// TwinCAT 3 PLC project Libraries
// Title: Logging/file library
// Company: Ziga
// Author: Ziga
// ProjectVersion: 0.0.1.1
// Description: A library containing file/logging functionalities.
// ProgramVersion: 3.1.4024.0
// libraries:
//   Tc2_Standard, * (Beckhoff Automation GmbH)
//   Tc2_System, * (Beckhoff Automation GmbH)
//   Tc2_Utilities, * (Beckhoff Automation GmbH)
//   Tc3_Module, * (Beckhoff Automation GmbH)
//   TcUnit, * (www.tcunit.org)
//   Core, * (Ziga)
// project tree:
//   SOURCE/FileHandler/POUs/ FB_FileHandler.TcPOU, I_FileHandler.TcIO (not stored)
//   SOURCE/Logger/DUTs/ E_LoggerState.TcDUT (not stored)
//   SOURCE/Logger/POUs/ FB_Logger.TcPOU
//   / TestsTask.TcTTO (not stored)
//   TESTS/ PRG_TESTS.TcPOU (not stored)
//   TESTS/Test suites/ FB_FileHandler_Tests.TcPOU (not stored), FB_Logger_Tests.TcPOU
//   Version/ Global_Version.TcGVL (not stored)
// real-time tasks:
//   TASK TestsTask: cycle T#10ms, priority 20, ADS port 350

// ---- SOURCE/FileHandler/POUs/FB_FileHandler.TcPOU
// A function block containing multiple file handling methods.
// For examples refer to tests in the folder "TESTS/Test suites", file "FB_FileHandlerTests".
FUNCTION_BLOCK FB_FileHandler EXTENDS ZigasLibs_Core.FB_ErrorSource IMPLEMENTS I_FileHandler

VAR
	_fileHandle		: UINT;
	_fileProperties	: ZigasLibs_Core.ST_FileProperties;
	_error			: BOOL;
	_amsAddress		: Tc2_System.ST_AmsAddr;
END_VAR

{attribute 'monitoring':='variable'}
(* Gets or sets the Ams address structure*)
PROPERTY AmsAddress : REFERENCE TO ZigasLibs_Core.Tc2_System.ST_AmsAddr
GET
AmsAddress ref= _amsAddress;
END_GET
SET
_amsAddress := AmsAddress;
END_SET
END_PROPERTY

(* Closes the file (if opened). Returns TRUE when done - method needs to be called until it returns TRUE!*)
METHOD PRIVATE Close : BOOL

VAR_INST
	fbFileClose			: Tc2_System.FB_FileClose;
	nCloseFileState		: UINT;
END_VAR

VAR CONSTANT
	FILE_CLOSE_START 		: UINT := 0;
	FILE_CLOSE_WAIT_BUSY	: UINT := 10;
	FILE_CLOSE_DONE			: UINT := 20;
END_VAR
IF THIS^.HandleCreated = FALSE THEN
	Close := TRUE;
	RETURN;
END_IF

_error := _error OR fbFileClose.bError;

CASE nCloseFileState OF
	FILE_CLOSE_START:
		fbFileClose(bExecute := FALSE);
		fbFileClose(bExecute := TRUE, hFile := _fileHandle);
		nCloseFileState := FILE_CLOSE_WAIT_BUSY;
		
	FILE_CLOSE_WAIT_BUSY:
		fbFileClose(bExecute := FALSE);
		IF NOT fbFileClose.bBusy AND NOT fbFileClose.bError THEN
			nCloseFileState := FILE_CLOSE_DONE;
		END_IF

	FILE_CLOSE_DONE:
		Close := TRUE;
		_fileHandle := 0;
		nCloseFileState := FILE_CLOSE_START;
END_CASE

_error := _error OR fbFileClose.bError;
IF fbFileClose.bError THEN
	_errorSource.ErrorCode := fbFileClose.nErrId;
END_IF
END_METHOD

(* Creates the file. Returns TRUE when done - method needs to be called until it returns TRUE!*)
METHOD Create : BOOL
VAR_INPUT
	(* If file already exists, it will be deleted and crated once again (content will be lost!)*)
	bOverwrite	: BOOL;
END_VAR

VAR_INST
	nFileCreateState	: UINT;
END_VAR

VAR CONSTANT
	FILE_CREATE_STATE_START					: UINT := 0;
	FILE_CREATE_STATE_OVERWRITE_OR_CREATE	: UINT := 10;
	FILE_CREATE_STATE_WAIT_DONE				: UINT := 20;
	FILE_CREATE_STATE_DONE					: UINT := 30;
END_VAR
CASE nFileCreateState OF
	FILE_CREATE_STATE_START:
		nFileCreateState := FILE_CREATE_STATE_OVERWRITE_OR_CREATE;
		
	FILE_CREATE_STATE_OVERWRITE_OR_CREATE:
		IF bOverwrite THEN
			IF THIS^.Open(mode := ZigasLibs_Core.E_FileOpenMode.BINARY_READ_WRITE_OVERWRITE_EXISTING) THEN
				nFileCreateState := FILE_CREATE_STATE_WAIT_DONE;
			END_IF
		ELSE
			IF THIS^.Open(mode := ZigasLibs_Core.E_FileOpenMode.BINARY_APPEND) THEN
				nFileCreateState := FILE_CREATE_STATE_WAIT_DONE;
			END_IF
		END_IF
		
	FILE_CREATE_STATE_WAIT_DONE:
		IF THIS^.Close() THEN
			nFileCreateState := FILE_CREATE_STATE_DONE;
		END_IF

	FILE_CREATE_STATE_DONE:
		nFileCreateState := FILE_CREATE_STATE_START;
END_CASE
END_METHOD

(* Deletes the file, if it exists. Returns TRUE when done - method needs to be called until it returns TRUE!*)
METHOD Delete : BOOL

VAR_INST
	fbFileDelete		: Tc2_System.FB_FileDelete;
	FtrigDeleteFinished	: Tc2_Standard.F_TRIG;
	bCheckIfFileExists	: BOOL;
	bFileExists			: BOOL;
END_VAR
fbFileDelete(
	bExecute := NOT fbFileDelete.bBusy,
	sPathName := ZigasLibs_Core.FileHelper.CreateFilePath(_fileProperties.FileLocation, _fileProperties.FileName,  ''));
	
FtrigDeleteFinished(CLK := fbFileDelete.bBusy);
IF FtrigDeleteFinished.Q THEN
	fbFileDelete(bExecute := FALSE);
	Delete := TRUE;
END_IF

_error := _error OR fbFileDelete.bError;
END_METHOD

{attribute 'monitoring':='variable'}
(* Gets the error state, if any of the functions failed.*)
PROPERTY Error : BOOL
GET
Error := _error;
END_GET
END_PROPERTY

(* Checks if the file exists. Returns TRUE when done - method needs to be called until it returns TRUE!*)
METHOD Exists : BOOL
VAR_INPUT
	(* When mehod is finished, the variable provided here will have the result, TRUE if file exists, FALSE if not.*)
	refFileExists	: REFERENCE TO BOOL;
END_VAR

VAR_INST
	fbFileExists			: Tc2_Utilities.FB_EnumFindFileEntry := (tTimeout := T#5S);
	nCheckFileExistState	: UINT;
END_VAR

VAR CONSTANT
	FILE_EXIST_STATE_PREPARE	: UINT := 0;
	FILE_EXIST_STATE_START		: UINT := 10;
	FILE_EXIST_STATE_CHECK		: UINT := 20;
	FILE_EXIST_STATE_DONE		: UINT := 30;
	FILE_EXIST_STATE_ERROR		: uint := 9999;
END_VAR
CASE nCheckFileExistState OF
	FILE_EXIST_STATE_PREPARE:
		fbFileExists(bExecute := FALSE, eCmd := Tc2_Utilities.E_EnumCmdType.eEnumCmd_First);
		refFileExists := FALSE;
		nCheckFileExistState := FILE_EXIST_STATE_START;
		
	FILE_EXIST_STATE_START:
		fbFileExists(bExecute := TRUE,
			sPathName := ZigasLibs_Core.FileHelper.CreateFilePath(_fileProperties.FileLocation, _fileProperties.FileName, ''),
			sNetId := ZigasLibs_Core.AmsHelper.NetIdToString(_amsAddress.netId));
		nCheckFileExistState := FILE_EXIST_STATE_CHECK;
	
	FILE_EXIST_STATE_CHECK:
		fbFileExists(bExecute := FALSE);
		IF NOT fbFileExists.bBusy THEN
			IF NOT fbFileExists.bError THEN
				IF fbFileExists.stFindFile.sFileName = _fileProperties.FileName THEN
					refFileExists := TRUE;
					nCheckFileExistState := FILE_EXIST_STATE_DONE;
				END_IF	
				IF NOT fbFileExists.bEOE THEN
					fbFileExists.eCmd := Tc2_Utilities.E_EnumCmdType.eEnumCmd_Next;
				ELSE
					refFileExists := FALSE;
					nCheckFileExistState := FILE_EXIST_STATE_DONE;
				END_IF
			ELSE
				nCheckFileExistState := FILE_EXIST_STATE_ERROR;
			END_IF
		END_IF
	
	FILE_EXIST_STATE_DONE:
		Exists := TRUE;
		nCheckFileExistState := FILE_EXIST_STATE_PREPARE;
		
	FILE_EXIST_STATE_ERROR:
		_errorSource.ErrorCode := fbFileExists.nErrID;
		nCheckFileExistState := FILE_EXIST_STATE_DONE;
		refFileExists := FALSE;
END_CASE

_error := _error OR fbFileExists.bError;
END_METHOD

{attribute 'monitoring':='variable'}
(* Gets or sets various file properties*)
PROPERTY FileProperties : REFERENCE TO ZigasLibs_Core.ST_FileProperties
GET
FileProperties ref= _fileProperties;
END_GET
SET
_fileProperties := FileProperties;
END_SET
END_PROPERTY

(* Gets the state of the file handle - if file is opened and handle is created returns TRUE.*)
PROPERTY PRIVATE HandleCreated : BOOL
GET
HandleCreated := _fileHandle <> 0;
END_GET
END_PROPERTY

(* Opens the file. Returns TRUE when done - method needs to be called until it returns TRUE!*)
METHOD PRIVATE Open : BOOL
VAR_INPUT
	mode	: ZigasLibs_Core.E_FileOpenMode;	// Mode in which the file is opened
END_VAR

VAR_INST
	fbFileOpen	: Tc2_System.FB_FileOpen;
END_VAR
IF THIS^.HandleCreated THEN
	Open := TRUE;
	RETURN;
END_IF

fbFileOpen(
	bExecute := NOT fbFileOpen.bBusy,
	sPathName := ZigasLibs_Core.FileHelper.CreateFilePath(_fileProperties.FileLocation, _fileProperties.FileName, ''),
	sNetId :=  ZigasLibs_Core.AmsHelper.NetIdToString(_amsAddress.netId),
	nMode := mode,
	hFile => _fileHandle);
	
_error := _error OR fbFileOpen.bError;	
IF fbFileOpen.bError THEN
	_errorSource.ErrorCode := fbFileOpen.nErrId;
END_IF
END_METHOD

(* Reads the content of the opened file to the target buffer.
 Returns TRUE when done - method needs to be called until it returns TRUE!*)
METHOD Read : BOOL
VAR_INPUT
	(* Pointer to the buffer, where the file content will be read to.*)
	ptrBuffer	: PVOID;
	(* Size of the buffer - SIZEOF()*)
	nBufferSize	: UDINT;
END_VAR


VAR_INST
	fbFileRead	: Tc2_System.FB_FileRead;
	nReadState	: UINT;
END_VAR

VAR CONSTANT
	READ_STATE_OPEN		: UINT := 0;
	READ_STATE_START	: UINT := 10;
	READ_STATE_WAIT		: UINT := 20;
	READ_STATE_DONE		: UINT := 30;
	READ_STATE_ERROR	: uint := 9999;
END_VAR
// An error is triggered if handle is not created or buffer pointer is invalid
IF ptrBuffer = 0 OR nBufferSize = 0 THEN
	_error := TRUE;
	Read := TRUE;
	RETURN;
END_IF

CASE nReadState OF
	READ_STATE_OPEN:
		IF THIS^.Open(mode := E_FileOpenMode.BINARY_READ) THEN
			nReadState := READ_STATE_START;
		END_IF	

	READ_STATE_START:
		fbFileRead(bExecute := FALSE);
		fbFileRead(
			bExecute := TRUE,
			hFile := _fileHandle,
			pReadBuff := ptrBuffer,
			cbReadLen := nBufferSize);
			
		nReadState := READ_STATE_WAIT;
		
	READ_STATE_WAIT:
		fbFileRead(bExecute := FALSE);
		IF fbFileRead.bError THEN
			nReadState := READ_STATE_ERROR;
		ELSIF fbFileRead.bBusy = FALSE THEN
			IF THIS^.Close() THEN
				nReadState := READ_STATE_DONE;
			END_IF
		END_IF	

	READ_STATE_DONE:
		Read := TRUE;
		nReadState := READ_STATE_OPEN;
		
	READ_STATE_ERROR:
		nReadState := READ_STATE_DONE;
		_errorSource.ErrorCode := fbFileRead.nErrId;
END_CASE

_error := _error OR fbFileRead.bError;
END_METHOD

METHOD PRIVATE WriteBinary : BOOL
VAR_INPUT
	ptrSource	: POINTER TO BYTE;	// Pointer to the source to be written - use ADR().
	nSize		: UDINT;	// Size of the source variable - use SIZEOF().
	mode		: E_FileOpenMode;
END_VAR

VAR_INST
	fbFileWrite	: Tc2_System.FB_FileWrite;
	nWriteState	: UINT;
END_VAR

VAR CONSTANT
	WRITE_OPEN_FILE	: UINT := 0;
	WRITE_START 	: UINT := 10;
	WRITE_WAIT_DONE	: UINT := 20;
	WRITE_DONE		: UINT := 30;
END_VAR
CASE nWriteState OF
	WRITE_OPEN_FILE:
		IF THIS^.Open(mode := mode) THEN
			nWriteState := WRITE_START;
		END_IF

	WRITE_START:
		fbFileWrite(bExecute := FALSE);
		fbFileWrite(
			bExecute := TRUE,
			hFile := _fileHandle,
			pWriteBuff := ptrSource,
			cbWriteLen := nSize);
			
		nWriteState := WRITE_WAIT_DONE;
	
	WRITE_WAIT_DONE:
		fbFileWrite(bExecute := FALSE);
		IF NOT fbFileWrite.bBusy THEN
			IF THIS^.Close() THEN
				nWriteState := WRITE_DONE;
			END_IF
		END_IF 
	
	WRITE_DONE:
		WriteBinary := TRUE;
END_CASE

_error := _error OR fbFileWrite.bError;

IF fbFileWrite.bError THEN
	_errorSource.ErrorCode := fbFileWrite.nErrId;
END_IF
END_METHOD

// Writes the content to the end of the file (appends).
// Returns TRUE when done - method needs to be called until it returns TRUE!
METHOD WriteBinary_Append : BOOL
VAR_INPUT
	ptrSource	: POINTER TO BYTE;	// Pointer to the source to be written - use ADR().
	nSize		: UDINT;	// Size of the source variable - use SIZEOF().
END_VAR
WriteBinary_Append := THIS^.WriteBinary(
	nSize := nSize, 
	ptrSource := ptrSource, 
	mode := E_FileOpenMode.BINARY_APPEND);
END_METHOD

(* Writes the content to the the file (overwrites any existing content).
 Returns TRUE when done - method needs to be called until it returns TRUE!*)
METHOD WriteBinary_Overwrite : BOOL
VAR_INPUT
	(* Pointer to the source to be written - use ADR().*)
	ptrSource	: POINTER TO BYTE;
	(* Size of the source variable - use SIZEOF().*)
	nSize	: UDINT;
END_VAR
WriteBinary_Overwrite := THIS^.WriteBinary(
	nSize := nSize, 
	ptrSource := ptrSource, 
	mode := E_FileOpenMode.BINARY_READ_WRITE_OVERWRITE_EXISTING);
END_METHOD

METHOD PRIVATE WriteLine : BOOL
VAR_INPUT
	(* Text to be written.*)
	sContent	: Tc2_System.T_MaxString;
	mode		: E_FileOpenMode;
END_VAR

VAR_INST
	fbFilePuts		: Tc2_System.FB_FilePuts;
	nWriteLineState	: UINT;
END_VAR

VAR CONSTANT
	WRITE_LINE_STATE_OPEN	: UINT := 0;
	WRITE_LINE_STATE_WRITE	: UINT := 10;
	WRITE_LINE_STATE_CLOSE	: UINT := 20;
	WRITE_LINE_STATE_DONE	: UINT := 30;
END_VAR
CASE nWriteLineState OF
	WRITE_LINE_STATE_OPEN:
		IF THIS^.Open(mode := mode) THEN
			nWriteLineState := WRITE_LINE_STATE_WRITE;
			fbFilePuts(bExecute := FALSE);
			fbFilePuts(
				bExecute := TRUE,
				hFile := _fileHandle,
				sLine := sContent,
				sNetId := ZigasLibs_Core.AmsHelper.NetIdToString(_amsAddress.netId),
				tTimeout := T#2S);
		END_IF
	
	WRITE_LINE_STATE_WRITE:
		fbFilePuts(bExecute := FALSE);
		IF fbFilePuts.bBusy = FALSE THEN
			nWriteLineState := WRITE_LINE_STATE_CLOSE;
		END_IF
	
	WRITE_LINE_STATE_CLOSE:
		IF THIS^.Close() THEN
			nWriteLineState := WRITE_LINE_STATE_DONE;
		END_IF
	
	WRITE_LINE_STATE_DONE:
		WriteLine := TRUE;
		nWriteLineState := WRITE_LINE_STATE_OPEN;
END_CASE

_error := _error OR fbFilePuts.bError;
IF fbFilePuts.bError THEN
	_errorSource.ErrorCode := fbFilePuts.nErrId;
END_IF
END_METHOD

// Writes the string content to the end of the file (appends). If the file does not exist, it will be created.
// Returns TRUE when done - method needs to be called until it returns TRUE!
METHOD WriteLine_Append : BOOL
VAR_INPUT
	(* Text to be written.*)
	sContent	: Tc2_System.T_MaxString;
END_VAR
WriteLine_Append := THIS^.WriteLine(
	sContent := sContent, 
	mode := E_FileOpenMode.TEXT_APPEND);
END_METHOD

(* Writes the string content to file and overwrites any existing content. If the file does not exist, it will be created.
 Returns TRUE when done - method needs to be called until it returns TRUE!*)
METHOD WriteLine_Overwrite : BOOL
VAR_INPUT
	(* Text to be written.*)
	sContent	: Tc2_System.T_MaxString;
END_VAR
WriteLine_Overwrite := THIS^.WriteLine(
	sContent := sContent,
	mode := E_FileOpenMode.TEXT_APPEND);
END_METHOD

END_FUNCTION_BLOCK

// ---- SOURCE/Logger/POUs/FB_Logger.TcPOU
FUNCTION_BLOCK FB_Logger IMPLEMENTS ZigasLibs_Core.I_LoggerEx
VAR
	_fileProperties			: ST_FileProperties;
	_logLevelHeaders		: ZigasLibs_Core.ST_LogLevelHeaders;
	_fileHandler			: FB_FileHandler;
	_events					: ARRAY[0..100] OF Tc2_System.T_MaxString;
	_state					: E_LoggerState;
	_fileExists				: BOOL;
	_localSystemTime		: ZigasLibs_Core.FB_LocalSystemTimeProvider;
	_localSystemTimeString	: Tc2_System.T_MaxString;
	_stringBuilder			: ZigasLibs_Core.FB_StringBuilderBase;
	_bufferFull				: BOOL;
	_amsAddress				: Tc2_System.ST_AmsAddr;
END_VAR

_localSystemTime();
_localSystemTimeString := _localSystemTime.CurrentTimeToString(
	dateSeperator := '.',
	fillWithZeros := TRUE,
	IncludeMilliseconds := FALSE,
	timeFormat := ZigasLibs_Core.E_TimeFormat.YYMMDD_HHMMSS,
	timeOfDaySeperator := ':');

IF _fileHandler.Error THEN
	_state := E_LoggerState.Error;
END_IF

CASE _state OF 
	E_LoggerState.IDLE:
		IF _events[0] <> '' AND _localSystemTime.CurrentTime.IsValid THEN
			_state := E_LoggerState.WRITE_TO_FILE;
		END_IF		
		
	E_LoggerState.WRITE_TO_FILE:
		_fileHandler.FileProperties.FileLocation := _fileProperties.FileLocation;
		_fileHandler.AmsAddress.netId := AmsAddress.netId;
		_fileHandler.FileProperties.FileName := _stringBuilder.Reset()
			.AddString(str := _fileProperties.FileName)
			.AddString(str := TimeForLogName())
			
		
		IF _fileHandler.WriteLine_Append(sContent := _events[0]) AND _fileHandler.Error = FALSE THEN
			THIS^.RemoveEvent();
			_state := E_LoggerState.IDLE;
		END_IF
		
	E_LoggerState.ERROR:
	
END_CASE

METHOD PRIVATE AddLogEntry
VAR_INPUT
	message	: Tc2_System.T_MaxString;
END_VAR

VAR
	i				: ZigasLibs_Core.T_ArrayIndexer;
	eventsMaxIndex	: ZigasLibs_Core.T_ArrayIndexer;
END_VAR
ZigasLibs_Core.ArrayHelper.SetAtFirstEmptySlot(
	arr := _events,
	item := message);

IF _events[100] <> '' THEN
	_bufferFull := TRUE;
ELSE
	_bufferFull := FALSE;
END_IF
END_METHOD

{warning 'add property implementation'}
(* Gets or sets the Ams address structure*)
PROPERTY AmsAddress : REFERENCE TO ZigasLibs_Core.Tc2_System.ST_AmsAddr
GET
AmsAddress ref= _amsAddress;
END_GET
SET
_amsAddress := AmsAddress;
END_SET
END_PROPERTY

PROPERTY PUBLIC BufferFull : BOOL
GET
BufferFull := _bufferFull;
END_GET
END_PROPERTY

(* Gets or set file properties.*)
PROPERTY FileProperties : REFERENCE TO ZigasLibs_Core.ST_FileProperties
GET
FileProperties REF= _fileProperties;
END_GET
SET
_fileProperties := FileProperties;
END_SET
END_PROPERTY

(* Logs the message without any additions.*)
METHOD LogDefault
VAR_INPUT
	message	: ZigasLibs_Core.Tc2_System.T_MaxString;
END_VAR
AddLogEntry(_stringBuilder.Reset() 
	.AddString(str := _localSystemTimeString)
	.AddString(str := ': ')
	.AddString(str := message)
	.Create());
END_METHOD

(* Logs the message by adding the error header to the start.*)
METHOD LogError
VAR_INPUT
	message	: ZigasLibs_Core.Tc2_System.T_MaxString;
END_VAR
AddLogEntry(_stringBuilder.Reset() 
	.AddString(str := _localSystemTimeString)
	.AddString(str := ': ')
	.AddString(str := _logLevelHeaders.Error)
	.AddString(str := message)
	.Create());
END_METHOD

(* Logs the message by adding the info header to the start.*)
METHOD LogInfo
VAR_INPUT
	message	: ZigasLibs_Core.Tc2_System.T_MaxString;
END_VAR
AddLogEntry(_stringBuilder.Reset() 
	.AddString(str := _localSystemTimeString)
	.AddString(str := ': ')
	.AddString(str := _logLevelHeaders.Info)
	.AddString(str := message)
	.Create());
END_METHOD

(* Gets or sets the headers which are applied to logs for their coresponding log levels.*)
PROPERTY LogLevelHeaders : REFERENCE TO ZigasLibs_Core.ST_LogLevelHeaders
GET
LogLevelHeaders ref= _logLevelHeaders;
END_GET
SET
_logLevelHeaders := LogLevelHeaders;
END_SET
END_PROPERTY

(* Logs the message by adding the info header to the start.*)
METHOD LogWarning
VAR_INPUT
	message	: ZigasLibs_Core.Tc2_System.T_MaxString;
END_VAR
AddLogEntry(_stringBuilder.Reset() 
	.AddString(str := _localSystemTimeString)
	.AddString(str := ': ')
	.AddString(str := _logLevelHeaders.Warning)
	.AddString(str := message)
	.Create());
END_METHOD

METHOD RemoveLogEntry
ZigasLibs_Core.ArrayHelper.ShiftDown(
	arr := _events, 
	element := _events[0]);
END_METHOD

METHOD PRIVATE TimeForLogName : STRING
TimeForLogName :=_localSystemTime.CurrentTimeToString(
	timeFormat := ZigasLibs_Core.E_TimeFormat.YYMMDD_HHMMSS,
	timeOfDaySeperator := '_',
	dateSeperator := '',
	fillWithZeros := TRUE,
	IncludeMilliseconds := FALSE)
END_METHOD

END_FUNCTION_BLOCK

// ---- TESTS/Test suites/FB_Logger_Tests.TcPOU
FUNCTION_BLOCK FB_Logger_Tests EXTENDS FB_TestSuite
VAR_INPUT
END_VAR
VAR_OUTPUT
END_VAR
VAR
END_VAR

Test_LogError();
Test_LogWarning();
Test_LogInfo();
Test_LogGeneric();

METHOD Test_LogError
VAR_INPUT
END_VAR
END_METHOD

METHOD Test_LogGeneric
VAR_INPUT
END_VAR
END_METHOD

METHOD Test_LogInfo
VAR_INPUT
END_VAR
END_METHOD

METHOD Test_LogWarning
VAR_INPUT
END_VAR
END_METHOD

END_FUNCTION_BLOCK
